// TIA Portal V20 export
DATA_BLOCK "DB_NordSetPoint"   // DB35
// stored: Access Published, MemoryReserve 100, Namespace LineB1
   VAR
      Line : Struct
         B1 : Struct   // -(0 - 16000) -> (CW: 0 - 100%) || +(0 - 16000) (CCW: 0 - 100%) || freq. has been set via NORDCON
            Conveyor : Array[_.minB1.._.maxB1] of DInt;
         END_STRUCT;
      END_STRUCT;
   END_VAR
BEGIN
END_DATA_BLOCK
